// TwinCAT 3 PLC project Base
// ProgramVersion: 3.1.4022.4
// libraries:
//   Tc2_Standard, * (Beckhoff Automation GmbH)
//   Tc2_System, * (Beckhoff Automation GmbH)
//   Tc2_Utilities, * (Beckhoff Automation GmbH)
//   Tc3_IotCommunicator, * (Beckhoff Automation GmbH)
//   Tc3_JsonXml, * (Beckhoff Automation GmbH)
//   Tc3_Module, * (Beckhoff Automation GmbH)
// project tree:
//   DUTs/ E_JsonStates.TcDUT (not stored)
//   GVLs/ CELL_STATE.TcGVL (not stored), CELL_WORKING_STATES.TcGVL (not stored), CLAMP_STATE.TcGVL (not stored), CELL_ACTION_STATE.TcGVL, DATA_SERVICE_STATE.TcGVL (not stored), MHS_STATE.TcGVL
//   / PlcTask.TcTTO
//   POUs/ FB_VirtualCell.TcPOU, I_CELL.TcIO, FB_Cell.TcPOU, FB_Clamp.TcPOU, FB_ClampSimulated.TcPOU (not stored), FB_DataService.TcPOU, FB_InterfaceIO.TcPOU, FB_InterfaceSimulated.TcPOU (not stored), FB_MHS.TcPOU, ITF_Cell.TcIO (not stored), JsonSaxHandler.TcPOU (not stored), MAIN.TcPOU, POU.TcPOU, FB_VirtualCellIntWriter.TcPOU (not stored)
// real-time tasks:
//   TASK PlcTask: cycle T#10ms, priority 20, ADS port 350

CONFIGURATION Base
    RESOURCE PLC ON TwinCAT3
        TASK PlcTask(INTERVAL := T#10ms, PRIORITY := 20);
        PROGRAM MAIN WITH PlcTask : MAIN;
    END_RESOURCE
END_CONFIGURATION

// ---- GVLs/CELL_ACTION_STATE.TcGVL
{attribute 'qualified_only'}
VAR_GLOBAL
			
TYPE 
	CELL_ACTION_STATE: (e_ToStandby, e_Standby, e_ToLoadPos, e_LoadPos, e_ToStartabel, e_Startabel, e_ToRunning , e_Running, 
				e_ToUnLoadPos, e_UnLoadPos,e_Finished, e_ToEmergencyStop, e_EmergencyStop, e_ToEmergencyOff, e_EmergencyOff , e_ErrorNum);
	
	
				
END_TYPE


END_VAR

// ---- GVLs/MHS_STATE.TcGVL
{attribute 'qualified_only'}
VAR_GLOBAL
TYPE
	MHS_STATE: (e_IDLE, e_PGO_POS, e_PGET_WP, e_PWAIT_DOOR, e_PWAIT_CLAMP, e_PPUT_WP,e_PCLOSE_CLAMP , e_PLEAFE_MACHINE, 
				e_GGO_POS, e_GGET_WP, e_GWAIT_DOOR, e_GWAIT_CLAMP ,e_GCLOSE_CLAMP , e_GLEAFE_MACHINE, e_AKTION_FINISHED, e_ERROR);
END_TYPE	

END_VAR

// ---- POUs/I_CELL.TcIO
INTERFACE I_CELL

METHOD GetErrorString : STRING
VAR_INPUT
END_VAR
END_METHOD

METHOD GetName : STRING
VAR_INPUT
END_VAR
END_METHOD

METHOD GetState : INT
VAR_INPUT
END_VAR
END_METHOD

METHOD GetWorkpiece : DINT
VAR_INPUT
END_VAR
END_METHOD

METHOD IsDisassemblyCell : BOOL
VAR_INPUT
END_VAR
END_METHOD

METHOD IsError : BOOL
VAR_INPUT
END_VAR
END_METHOD

METHOD IsIdle : BOOL
VAR_INPUT
END_VAR
END_METHOD

METHOD IsVirtualCell : BOOL
VAR_INPUT
END_VAR
END_METHOD

METHOD RequestActionState : BOOL
VAR_INPUT
	csStateRequest : CELL_ACTION_STATE;
END_VAR
END_METHOD

METHOD RequestWork : BOOL
VAR_INPUT
END_VAR
END_METHOD

METHOD SetDisassemblyCell : BOOL
VAR_INPUT
	bIsDisassemblyCell : BOOL;
END_VAR
END_METHOD

METHOD SetGetDataServiceEnable : BOOL
VAR_INPUT
END_VAR
END_METHOD

METHOD SetName : BOOL
VAR_INPUT
	sName :string ;
END_VAR
END_METHOD

METHOD SetPutDataServiceEnable : BOOL
VAR_INPUT
END_VAR
END_METHOD

METHOD SetVirtualCell : BOOL
VAR_INPUT
END_VAR
END_METHOD

METHOD SetWorkpiece : BOOL
VAR_INPUT
	iWorkpiece : DINT;
	sWorkpieceID : STRING;
END_VAR
END_METHOD

METHOD StateMachine : BOOL
VAR_INPUT
END_VAR
END_METHOD

END_INTERFACE

// ---- POUs/MAIN.TcPOU

PROGRAM MAIN
	
VAR



// Allg. nitwendige Variablen
m_bInit : BOOL;
I : DINT;
sString : STRING;
diDint : DINT;
bBOOL:BOOL;
m_iCellUpdateIter : INT := 0; // Iterationsvariable für die Json Strings der Zelle

// Zellen
fbCellA2 : FB_Cell;
fbCellB2 : FB_Cell; 
fbCellB5 : FB_Cell; 
fbCellV1 : FB_VirtualCell;
fbCellV2 : FB_VirtualCell;

aCellList : ARRAY [1..5] OF I_CELL; // Liste der Zellen
m_iNumberOfCells : DINT := 5; // Bei hinzufügen/löschen einer Zelle ist hier die Anzahl anzupassen

// MHS 
fbMHS : FB_MHS;

// Kommunikations-Variabeln für Aktionen von der GUI


m_bTrigger : BOOL;// Trigger zum zyklischen Aktualisieren der Anwendung
m_iTriggerTimer : INT; // Zähler zum Trigger 
m_sJsonTrigger : STRING(80);

m_sActionID : STRING(80);
m_sWPID : STRING(80);
m_iWPRequest : DINT;
m_sCellRequest : STRING;
m_iActionRequest : DINT;
m_iActionState : DINT;


m_sActionIDLast : STRING(80);
m_sWPIDLast : STRING(80);
m_iWPRequestLast : DINT;
m_iCellRequestLast : DINT;
m_iActionRequestLast : DINT;
m_iActionStateLast : DINT;
m_iCellRequest : DINT;

m_bAktionInProgress : BOOL; 

//JSON-Variablen
	//Writer
	m_iJsonTimer 		: DINT;
 	dtTimestamp 		: DATE_AND_TIME := DT#2017-04-04-12:42:42;
 	fbJson      		: FB_JsonSaxWriter;
 	sJsonDocCells   	: STRING(3000);
	//Reader
 	fbJsonReader    		: FB_JsonSaxReader;
	pJsonParse 				: JsonSaxHandler;
	sJsonDocAction			: STRING(255);
	sJsonDocLastAction   : STRING(255);
	
	sJsonDocError 		 : STRING (255); 

END_VAR


//Initialisierung
IF NOT m_bInit THEN
	// Hier die FunktionsBlöcke der Maschinen in das Array Schreiben !!!
	aCellList[1] := fbCellA2;
	aCellList[1].SetName('A2'); // Geometrieerfassung
	//aCellList[1].SetPutDataServiceEnable();
	aCellList[2] := fbCellB2;
	aCellList[2].SetName('B2'); // Rekonturierng
 	aCellList[2].SetGetDataServiceEnable();
	aCellList[3] := fbCellB5;
	aCellList[3].SetName('B5'); // LaserSchweißen
	aCellList[3].SetGetDataServiceEnable();
	aCellList[3].SetPutDataServiceEnable();
	
	aCellList[4] := fbCellV1;
	aCellList[4].SetName('V1'); // Virtuell
	aCellList[4].SetVirtualCell();
	
	
	aCellList[5] := fbCellV2;
	aCellList[5].SetName('V2'); // Virtuell
	aCellList[5].SetVirtualCell();

	// Intitialisiert setzen 
	m_bInit := TRUE;

END_IF



IF m_bAktionInProgress = FALSE THEN 
	// Abfrage ob neue Aktion angestoßen wurde
	CheckForNewAction();
		
END_IF


//Zustandmaschinen
	// Zyklische aktualisierung der Zellen-Zustandsmaschinen
	I := 1;
	FOR I:=1 TO m_iNumberOfCells BY 1 DO
    	aCellList[I].StateMachine();
	END_FOR;
	// Zyklische aktualisierung der MHS-Zustandsmaschine
	fbMHS();
// Zustandsmaschinen durchgelaufen

IF m_bAktionInProgress THEN// MHS muss den Zustand der involvierten Zelle kennen und eine Zustand von der Zelle anfordern können
	
	fbMHS.SetStateCurrentMachineForAction( aCellList[fbMHS.GetCurrentCellForAction()].GetState());// Aktualisieren des MHS Zustandes
	IF fbMHS.NeededCellStatePending() THEN // Wenn das MHS einen Zellenzustand verlangt wird er folgend übergeben
		aCellList[fbMHS.GetCurrentCellForAction()].RequestActionState(fbMHS.SendNeededToCell() );// Übergabe des geforderten Zellenzustandes an die Zelle
	END_IF
END_IF


// Abfrage ob letzte Aktion Abgeschlossen wurde.... auf WIN abgefragen um neue Aktion zu senden 
IF fbMHS.GetActionFinished() THEN
	m_bAktionInProgress := FALSE; 
	IF m_iActionRequestLast = 2 THEN // Bestuecken
		aCellList[m_iCellRequestLast].SetWorkpiece(m_iWPRequestLast, m_sWPIDLast);// Werkstück an die Zelle übergeben
		aCellList[m_iCellRequestLast].RequestWork(); // Starten der Bearbeitung in der Zelle		
	ELSE
		aCellList[m_iCellRequestLast].SetWorkpiece(0, 'Empty'); // Werkstück der Zelle nehmen
	END_IF
	m_iActionStateLast := 3;
END_IF

// Schreiben der JSON-Strings zur Kommunikation der Systemdemostrator-Anwendung
WriteJsonStrings();

METHOD CheckForNewAction : BOOL
VAR_INPUT
END_VAR
	 ParseNewAction();
	m_iCellRequest := NumberOfCellName(m_sCellRequest);
	IF	 (NOT(m_sActionID = m_sActionIDLast)) AND (m_iCellRequest <= m_iNumberOfCells) AND (m_iCellRequest > 0) THEN // Neue Aktion und Zelle ist existent
		IF NOT(aCellList[m_iCellRequest].IsVirtualCell())THEN
			
			IF aCellList[m_iCellRequest].IsIdle() THEN // Zelle frei
				// Neue Aktion an das MHS übergeben 
				WriteNewActionToMHS();
				m_bAktionInProgress := TRUE;// Setzen des Flags 
			END_IF
		ELSE // Im Falle einer Aktion für eine virtuelle Zelle
			IF aCellList[m_iCellRequest].IsIdle() THEN
				aCellList[m_iCellRequest].SetWorkpiece(0, m_sWPID );
				aCellList[m_iCellRequest].RequestWork();	
				//m_iActionStateLast := 3; // Wird nur angestoßen ist direkt fertig mit der Aktion, so dass eine weitere beginnen kann.
			END_IF
		END_IF
	
	END_IF
END_METHOD

METHOD NumberOfCellName : DINT
VAR_INPUT
	sNameOfCell : STRING;
END_VAR
FOR I:=1 TO m_iNumberOfCells BY 1 DO
    IF sNameOfCell = aCellList[I].GetName() THEN
		NumberOfCellName :=I;
	END_IF
END_FOR;
END_METHOD

METHOD ParseNewAction : BOOL
VAR_INPUT
END_VAR

	// Aktion JSonDoc Lesen des Aktuellen Strings
	fbJsonReader.Parse( sJson := sJsonDocAction, ipHdl := pJsonParse);
	
	IF pJsonParse.IsFinished() THEN
		// Übergabe der geparsten Variablen
		m_sActionID	:=	pJsonParse.GetActionID();
		m_sWPID	:=	pJsonParse.GetWPID();
		m_iWPRequest := pJsonParse.GetWPPlace(); 
		m_sCellRequest := pJsonParse.GetCell(); 
		m_iActionRequest:=pJsonParse.GetActionType();
		
		// Für den nächsten Durchlauf zurücksetzen 
		pJsonParse.Reset();
	ELSE
		// Parsen des Json-Strings
		fbJsonReader.Parse( sJson := sJsonDocAction, ipHdl := pJsonParse);
	END_IF
END_METHOD

METHOD WriteJSonDocAction : BOOL
VAR_INPUT
END_VAR

fbJson.ResetDocument();
		//fbJson.StartArray();
fbJson.StartObject();
            fbJson.AddKey('m_sActionID');
			fbJson.AddString(m_sActionIDLast);
            fbJson.AddKey('m_sWPID');
			sString := m_sWPIDLast;
			fbJson.AddString(sString);
            fbJson.AddKey('m_iWPPlace');
			fbJson.AddDint(m_iWPRequestLast);
            fbJson.AddKey('m_sCell');
			IF m_iCellRequestLast > 0 THEN// Sonst würden das Zell Array außerhalb seines Bereiches angesproehcen werden
				sString := aCellList[m_iCellRequestLast].GetName();
			ELSE
				sString := 'EmptyAction';				
			END_IF
			fbJson.AddString(sString);
            fbJson.AddKey('m_eActionType');
			fbJson.AddDint(m_iActionRequestLast);
            fbJson.AddKey('m_iActionState');
			fbJson.AddDint(m_iActionStateLast);	
fbJson.EndObject();
	sJsonDocLastAction := fbJson.GetDocument();

WriteJSonDocAction := TRUE;
END_METHOD

METHOD WriteJSonDocCells : BOOL
VAR_INPUT
END_VAR
// Merken alle Zellen einzelnd Updaten, weil es nicht möglich ist die über 255 Zeichen langen Strings aller zu übertragen

	fbJson.ResetDocument();
	//fbJson.StartObject();
	//fbJson.AddKey('Timestamp');
	
	//fbJson.AddDateTime(dtTimestamp);
	m_iCellUpdateIter := m_iCellUpdateIter +1 ; 
	IF m_iCellUpdateIter > m_iNumberOfCells THEN
		m_iCellUpdateIter := 1;
	END_IF
		//fbJson.AddKey('Cell');
		m_sActionIDLast := m_sActionID;
		m_iWPRequestLast := m_iWPRequest; 		
		m_iCellRequestLast := m_iCellRequest;
		m_iActionRequestLast :=	m_iActionRequest;
		fbJson.StartObject();
		//fbJson.StartArray();
		fbJson.AddKey('Name');
		sString := aCellList[m_iCellUpdateIter].GetName();
		fbJson.AddString(sString);
		fbJson.AddKey('State');
		fbJson.AddDint(aCellList[m_iCellUpdateIter].GetState());
		fbJson.AddKeyBool('Idle',aCellList[m_iCellUpdateIter].IsIdle());
		fbJson.AddKey('Workpiece');
		fbJson.AddDint(aCellList[m_iCellUpdateIter].GetWorkpiece());
		fbJson.AddKey('IsDisassemblyCell');
		fbJson.AddBool(aCellList[m_iCellUpdateIter].IsDisassemblyCell());
		fbJson.AddKey('IsVirtualCell');
		fbJson.AddBool(aCellList[m_iCellUpdateIter].IsVirtualCell());
		fbJson.EndObject();
		
		

	
	
	//fbJson.EndObject();
	sJsonDocCells := '';
	sJsonDocCells := fbJson.GetDocument();
	
WriteJSonDocCells := TRUE;
END_METHOD

METHOD WriteJSonError : BOOL
VAR_INPUT
END_VAR
	fbJson.ResetDocument();


	I := 1;
	FOR I:=1 TO m_iNumberOfCells BY 1 DO
		IF aCellList[I].IsError() THEN
			fbJson.StartObject();
			fbJson.AddKey('Name');
			sString := aCellList[I].GetName();
			fbJson.AddString(sString);	
			fbJson.AddKey('Workpiece');
			fbJson.AddDint(aCellList[I].GetWorkpiece());
			fbJson.AddKey('Error');
			sString := aCellList[I].GetErrorString();
			fbJson.AddString(sString);
			fbJson.EndObject();	
			
			sJsonDocError := '';
			sJsonDocError := fbJson.GetDocument();

		END_IF	
	
	END_FOR;
END_METHOD

METHOD WriteJsonStrings : BOOL
VAR_INPUT
END_VAR




// Erstellen eines Json-Strings für die GUI alle 100 Durchläufe 0,1s
m_iJsonTimer := m_iJsonTimer+1;
IF m_iJsonTimer > 150 THEN
	WriteJSonDocCells();
	WriteJSonDocAction();
	
	m_iJsonTimer := 0;
	
END_IF
// GUI Trigger um zyklische Aufrufe auch bei nicht veränderten JSON-Strings zu erzielen
// Ohne den Trigger würde ine Prüfung des Regenerationspfades bei nicht mehr vorhanden Aktion im Pfad nicht fortgeführt werden
IF m_iTriggerTimer > 2500 THEN
	m_bTrigger :=  NOT(m_bTrigger);// Bool abwechselnd false und true
	WriteJsonTrigger();
	m_iTriggerTimer := 0; 
END_IF
	
m_iTriggerTimer := m_iTriggerTimer + 1;
END_METHOD

METHOD WriteJsonTrigger : BOOL
VAR_INPUT
END_VAR
fbJson.ResetDocument();
		//fbJson.StartArray();
fbJson.StartObject();
            fbJson.AddKey('m_bTrigger');
			fbJson.AddBool(m_bTrigger);
fbJson.EndObject();
	m_sJsonTrigger := fbJson.GetDocument();
END_METHOD

METHOD WriteNewActionToMHS : BOOL
VAR_INPUT
END_VAR
// Übergaben der neuen Aktion an das MHS
fbMHS.RequestAction(	iWorkpiece := m_iWPRequest, iCell := m_iCellRequest, bRequest := m_iActionRequest);
// Speichern des Zustandes
m_sActionIDLast := m_sActionID;
m_sWPIDLast := m_sWPID; 
m_iWPRequestLast := m_iWPRequest; 		
m_iCellRequestLast := m_iCellRequest;
m_iActionRequestLast :=	m_iActionRequest;

m_iActionStateLast := 2;
END_METHOD

END_PROGRAM

// ---- POUs/FB_Cell.TcPOU
FUNCTION_BLOCK FB_Cell IMPLEMENTS I_CELL
VAR_INPUT
	
END_VAR
VAR_OUTPUT
END_VAR
VAR
	m_csStateRequest : CELL_ACTION_STATE;
	m_csStateRequestOld : CELL_ACTION_STATE;
	m_csState : CELL_ACTION_STATE;
	m_csStateLastCycle : CELL_ACTION_STATE;
	m_csStateLastAction : CELL_ACTION_STATE;
	
	
	m_csSRWorkingState : CELL_WORKING_STATES := CELL_WORKING_STATES.e_FINISHED;
	m_csSRWorkingStateLast : CELL_WORKING_STATES := CELL_WORKING_STATES.e_FINISHED;
	// Eigenschaften
	m_sName : STRING;
	m_bIsDisassemblyCell : BOOL;
	
	
	m_iWorkpiece : DINT;
	m_sWorkpieceID : STRING;
	

	m_csCellState : CELL_STATE;
	m_csCellStateLast : CELL_STATE;

	fbInterface : FB_InterfaceSimulated;
	fbClamp : FB_ClampSimulated; 
	
	m_sErrorString : STRING;
	
	// DataServices
	
	fbDataServicePut : FB_DataService;
	m_bDataServicePutEnable : BOOL;
	fbDataServiceGet : FB_DataService;
	m_bDataServiceGetEnable : BOOL;
	m_sConfigString : STRING;
	m_sConfigStringEndGet : STRING  := '_Get.exe';
	m_sConfigStringEndPut : STRING  := '_Put.exe';
	m_sDataServiceDir: STRING  := 'C:\temp\Debug\';
	m_sDataServiceIP: STRING  := '192.168.178.24.1.1';
	
END_VAR

METHOD GetErrorString : STRING
VAR_INPUT
END_VAR
END_METHOD

METHOD GetName : STRING
VAR_INPUT
END_VAR
GetName := m_sName;
END_METHOD

METHOD PUBLIC GetState : INT
VAR_INPUT
	
END_VAR
GetState := m_csState;
END_METHOD

METHOD GetWorkpiece : DINT
VAR_INPUT
END_VAR
GetWorkpiece := m_iWorkpiece;
END_METHOD

METHOD IsDisassemblyCell : BOOL
VAR_INPUT
END_VAR
IsDisassemblyCell := m_bIsDisassemblyCell;
END_METHOD

METHOD IsError : BOOL
VAR_INPUT
END_VAR
IF m_csCellState = CELL_STATE.e_ERROR THEN
	IsError := TRUE;
END_IF
END_METHOD

METHOD IsIdle : BOOL
VAR_INPUT
END_VAR
IF m_csCellState = CELL_STATE.e_IDEL THEN
	IsIdle := TRUE;
END_IF
END_METHOD

METHOD IsVirtualCell : BOOL
VAR_INPUT
END_VAR
IsVirtualCell :=FALSE;
END_METHOD

METHOD PUBLIC RequestActionState : BOOL
VAR_INPUT
	csStateRequest : CELL_ACTION_STATE;
END_VAR
m_csStateRequest := csStateRequest;
END_METHOD

METHOD RequestWork : BOOL
VAR_INPUT
END_VAR
m_csCellState := CELL_STATE.e_WORKING;
END_METHOD

METHOD SetDisassemblyCell : BOOL
VAR_INPUT
	bIsDisassemblyCell : BOOL;
END_VAR
m_bIsDisassemblyCell := bIsDisassemblyCell;
END_METHOD

METHOD SetGetDataServiceEnable : BOOL
VAR_INPUT
END_VAR
m_bDataServiceGetEnable := TRUE;
SetGetDataServiceEnable := TRUE;
END_METHOD

METHOD SetName : BOOL
VAR_INPUT
	sName :string ;
END_VAR
m_sName := sName;
END_METHOD

METHOD SetPutDataServiceEnable : BOOL
VAR_INPUT
END_VAR
m_bDataServicePutEnable := TRUE;
SetPutDataServiceEnable := TRUE;
END_METHOD

METHOD SetVirtualCell : BOOL
VAR_INPUT
END_VAR
END_METHOD

METHOD SetWorkpiece : BOOL
VAR_INPUT
	iWorkpiece : DINT;
	sWorkpieceID : STRING;
END_VAR
m_iWorkpiece := iWorkpiece;
m_sWorkpieceID := sWorkpieceID;
END_METHOD

METHOD PUBLIC StateMachine : BOOL
VAR_INPUT
END_VAR

fbInterface();
fbClamp();



// Error-Abfragen
IF fbClamp.IsError() THEN
	m_csCellState := CELL_STATE.e_ERROR; 
	m_sErrorString := 'CLAMP-Error: Clamp is closed without Workpiece';
END_IF


//Zellen Zustandsmaschine

CASE m_csCellState OF 
	CELL_STATE.e_IDEL:
			
	
		;
 	CELL_STATE.e_MHS_ACTION;
		//SubRoutine für Aktion beim beladen aktuell leer da alles vom MHS gesteuert wird 
	
		;
	CELL_STATE.e_WORKING:
		//SubRoutine zum Durchführen einer Bearbeitung
		
		IF NOT (m_csCellStateLast = m_csCellState) THEN
			m_csSRWorkingState := CELL_WORKING_STATES.e_START;
			IF m_bDataServiceGetEnable THEN
				fbDataServiceGet.SetNetIP(m_sDataServiceIP);
				fbDataServiceGet.SetWorkingDirectory(m_sDataServiceDir);
				m_sConfigString := m_sDataServiceDir;
				m_sConfigString := CONCAT(m_sConfigString , m_sName); // erstellen des Pfades der Applikation 
				m_sConfigString := CONCAT(m_sConfigString , m_sConfigStringEndGet);
				fbDataServiceGet.SetCommandLine(m_sWorkpieceID);
				fbDataServiceGet.SetPathOfApplication(m_sConfigString);
				fbDataServiceGet.StartDataService();
			END_IF
		END_IF
			
		CASE m_csSRWorkingState OF
			
			CELL_WORKING_STATES.e_START:
				
				IF NOT (m_csSRWorkingStateLast = m_csSRWorkingState )THEN
					m_csStateRequest := CELL_ACTION_STATE.e_Startabel;
				END_IF
				
				
				IF m_csState = CELL_ACTION_STATE.e_Startabel AND (fbDataServiceGet.IsFinished() OR NOT(m_bDataServiceGetEnable) )  THEN // Zelle bereit zum Starten und DataServiceGet fertig oder nicht konfiguriert
					m_csSRWorkingState:= CELL_WORKING_STATES.e_WORKING;
					fbDataServiceGet.SetIdle();
					m_csStateRequest:= CELL_ACTION_STATE.e_Running;
				END_IF
				
				
			CELL_WORKING_STATES.e_WORKING:
				IF NOT (m_csSRWorkingStateLast = m_csSRWorkingState) THEN
					m_csStateRequest := CELL_ACTION_STATE.e_Running;
				END_IF
				
				IF m_csState = CELL_ACTION_STATE.e_Finished THEN
					m_csSRWorkingState := CELL_WORKING_STATES.e_FINISHED;
					IF m_bDataServicePutEnable THEN
						fbDataServicePut.SetNetIP('192.168.178.24.1.1');
						fbDataServicePut.SetWorkingDirectory('C:\temp\Debug');
						m_sConfigString := 'C:\temp\Debug\';						
						m_sConfigString := CONCAT(m_sConfigString , m_sName); // erstellen des Pfades der Applikation 
						m_sConfigString := CONCAT(m_sConfigString , m_sConfigStringEndPut);// erstellen des Pfades der Applikation
						fbDataServicePut.SetCommandLine(m_sWorkpieceID);
						fbDataServicePut.SetPathOfApplication(m_sConfigString);
						fbDataServicePut.StartDataService();
						m_csSRWorkingState := e_DATAPUT;
					END_IF
		
				END_IF
			CELL_WORKING_STATES.e_DATAPUT:
					IF fbDataServicePut.IsFinished() THEN
						fbDataServicePut.SetIdle();
						m_csSRWorkingState := CELL_WORKING_STATES.e_FINISHED;
					END_IF
					IF fbDataServicePut.IsError() THEN
						fbDataServicePut.SetIdle();
						m_csSRWorkingState := CELL_STATE.e_ERROR;
					END_IF
					
			CELL_WORKING_STATES.e_FINISHED:
				m_csCellState := CELL_STATE.e_IDEL;
			
		END_CASE
		
		
		
	CELL_STATE.e_ERROR:
		m_csState :=CELL_ACTION_STATE.e_ToEmergencyStop;
	
		
END_CASE
m_csSRWorkingStateLast := m_csSRWorkingState;
m_csCellStateLast := m_csCellState;

IF NOT (m_csStateRequestOld = m_csStateRequest) THEN
	m_csState := m_csStateRequest - 1;
	m_csStateRequestOld := m_csStateRequest;
END_IF


// Aktions Zustandsmaschine
CASE m_csState OF 
	CELL_ACTION_STATE.e_ToStandby:
		IF NOT (m_csStateLastCycle = m_csState) THEN
			fbInterface.SetStandby(TRUE);
			m_csStateLastAction := m_csStateLastCycle;
		END_IF
		
		IF fbInterface.GetStandby() THEN
			m_csState := e_Standby; 
		END_IF
		
	CELL_ACTION_STATE.e_Standby :
	
		IF NOT (m_csStateLastCycle = m_csState) THEN
			m_csStateLastAction := m_csStateLastCycle;
		END_IF
		fbInterface.SetStandby(FALSE);
		
	CELL_ACTION_STATE.e_ToLoadPos:
	
		IF NOT (m_csStateLastCycle = m_csState) THEN
			m_csStateLastAction := m_csStateLastCycle;
			fbInterface.SetMoveToLoad(TRUE);
			fbClamp.SetOpenClamp();
		END_IF
		
		IF fbInterface.GetLoadPos() AND fbClamp.IsOpen() THEN
			m_csState := e_LoadPos; 
		END_IF
		
		
	CELL_ACTION_STATE.e_LoadPos:
	
		IF NOT (m_csStateLastCycle = m_csState) THEN
			m_csStateLastAction := m_csStateLastCycle;
		END_IF
		fbInterface.SetMoveToLoad(FALSE);
				
		
	CELL_ACTION_STATE.e_ToStartabel:
	
		IF NOT (m_csStateLastCycle = m_csState) THEN
			m_csStateLastAction := m_csStateLastCycle;
			fbClamp.SetCloseClampFull();
		END_IF
		
		
		IF  fbClamp.IsClosedFull() THEN //fbInterface.GetStartable() AND
			m_csState := e_Startabel; 
		END_IF
		
	CELL_ACTION_STATE.e_Startabel:
	
		IF NOT (m_csStateLastCycle = m_csState) THEN
			m_csStateLastAction := m_csStateLastCycle;
			
		END_IF
		
	CELL_ACTION_STATE.e_ToRunning:
	
		IF NOT (m_csStateLastCycle = m_csState) THEN
			m_csStateLastAction := m_csStateLastCycle;
			fbInterface.SetStart(TRUE);
		END_IF
		
		IF fbInterface.GetIsRunning() THEN
			m_csState := CELL_ACTION_STATE.e_Running; 
		END_IF
		
	CELL_ACTION_STATE.e_Running:
	
		IF NOT (m_csStateLastCycle = m_csState) THEN
			m_csStateLastAction := m_csStateLastCycle;
		END_IF
		fbInterface.SetStart(FALSE);
		IF fbInterface.GetFinished() THEN
			m_csState := CELL_ACTION_STATE.e_Finished;		
		END_IF
	CELL_ACTION_STATE.e_Finished:
		IF NOT (m_csStateLastCycle = m_csState) THEN
			m_csStateLastAction := m_csStateLastCycle;
		END_IF
		
	CELL_ACTION_STATE.e_ToUnLoadPos:
 
		IF NOT (m_csStateLastCycle = m_csState) THEN
			m_csStateLastAction := m_csStateLastCycle;
			fbClamp.SetOpenClamp();
		END_IF
		
		
		IF fbInterface.GetUnloadPos() AND fbClamp.IsOpen() THEN
			m_csState := e_UnLoadPos; 
		END_IF
		
	CELL_ACTION_STATE.e_UnLoadPos:
	
		IF NOT (m_csStateLastCycle = m_csState) THEN
			m_csStateLastAction := m_csStateLastCycle;
		END_IF
		
	CELL_ACTION_STATE.e_ToEmergencyStop:
	
		IF NOT (m_csStateLastCycle = m_csState) THEN
			m_csStateLastAction := m_csStateLastCycle;
		END_IF
		
		
		IF fbInterface.GetEmergencyStop() THEN
			m_csState := e_EmergencyStop; 
		END_IF
		
	CELL_ACTION_STATE.e_EmergencyStop:
	
		IF NOT (m_csStateLastCycle = m_csState) THEN
			m_csStateLastAction := m_csStateLastCycle;
		END_IF
		
	CELL_ACTION_STATE.e_ToEmergencyOff:
	
		IF NOT (m_csStateLastCycle = m_csState) THEN
			m_csStateLastAction := m_csStateLastCycle;
		END_IF
		
		
		IF fbInterface.GetEmergencyStop() THEN
			m_csState := e_EmergencyOff; 
		END_IF
		
	CELL_ACTION_STATE.e_EmergencyOff:
	
		IF NOT (m_csStateLastCycle = m_csState) THEN
			m_csStateLastAction := m_csStateLastCycle;
		END_IF
		
	ELSE
		IF NOT (m_csStateLastCycle = m_csState) THEN
			m_csStateLastAction := m_csStateLastCycle;
		END_IF
		
END_CASE

IF m_bDataServiceGetEnable THEN
	fbDataServiceGet();
END_IF
IF m_bDataServicePutEnable THEN	
	fbDataServicePut();
END_IF

m_csStateLastCycle := m_csState;
END_METHOD

END_FUNCTION_BLOCK

// ---- POUs/FB_DataService.TcPOU
FUNCTION_BLOCK FB_DataService
VAR_INPUT
END_VAR
VAR_OUTPUT
END_VAR
VAR
	fbStartProcess : NT_StartProcess;

	m_sCommandLine : STRING;
	m_sNetIP : STRING;
	m_sWorkingdirektory : STRING;
	m_sPathOfApplication : STRING;
	m_bStart : BOOL;
	m_eState : DATA_SERVICE_STATE;
	m_sErrCode : STRING;
	m_iReturnValue : DINT;
END_VAR

fbStartProcess.NETID 		:= m_sNetIP; // IP Adresse des Rechners auf dem die Zwillinge liegen
fbStartProcess.COMNDLINE 	:= m_sCommandLine; // Hier muss die ZwillingsID/ ProjektID übertragen werden
fbStartProcess.DIRNAME 		:= m_sWorkingdirektory; // Dieser Verzeichnis ist  vermutlich immer c:\TEMP
fbStartProcess.PATHSTR 		:= m_sPathOfApplication; // Pfad direkt zur DataService.exe wobei sich diese aus dem Zell-Namen ergibt 


IF fbStartProcess.ERR THEN // Fehlerabrage bereits vor der Zustandsmaschine 
	m_eState := DATA_SERVICE_STATE.e_ERROR;
END_IF 


CASE m_eState OF 
	DATA_SERVICE_STATE.e_IDLE:
	
		IF  m_bStart = TRUE THEN
			fbStartProcess.START := TRUE;
			m_bStart := FALSE; //Nurpositive Flanke übergeben		
		END_IF
	
		IF fbStartProcess.BUSY = TRUE THEN // Wenn der Funktionsblock selber Busy meldet in den nächsten Zustand
			m_eState := DATA_SERVICE_STATE.e_BUSY;
			fbStartProcess.START := FALSE;  
		END_IF
		
	DATA_SERVICE_STATE.e_BUSY:
	
 		IF fbStartProcess.BUSY = FALSE THEN
			IF m_iReturnValue = 1 THEN // Übergabewert der DataService.exe
				m_iReturnValue := 0; // Zurücksetzen für den nächsten Durchlauf
				m_eState := DATA_SERVICE_STATE.e_FINISHED;
			END_IF
			IF m_iReturnValue = 2 THEN
				m_eState := DATA_SERVICE_STATE.e_ERROR; 					
			END_IF		
		END_IF 
		
	DATA_SERVICE_STATE.e_FINISHED: // Zustand erforderlich da somit ein Zyklus lang abgefragt werden kann ob der Ablauf erfolgreich war
			
 		
		
	DATA_SERVICE_STATE.e_ERROR:
	
		m_sErrCode := UDINT_TO_STRING (fbStartProcess.ERRID); // Der Fehler wird als ganzzahl in den String geschrieben 
	
ELSE // Sicherheit bei falschem Wert
		m_eState := DATA_SERVICE_STATE.e_ERROR;
		m_sErrCode := 'Falscher Wert DataService-Status nicht vorhanden';
		
END_CASE

// Aufruf des Funktionblocks NT_StartProcess
fbStartProcess();

METHOD GetErrorCode : STRING
VAR_INPUT
END_VAR

VAR
END_VAR
GetErrorCode :=m_sErrCode;
END_METHOD

METHOD IsBusy : BOOL
VAR_INPUT
END_VAR
IF m_eState = DATA_SERVICE_STATE.e_BUSY THEN
	IsBusy := TRUE;
END_IF
END_METHOD

METHOD IsError : BOOL
VAR_INPUT
END_VAR
IF m_eState = DATA_SERVICE_STATE.e_ERROR THEN
	IsError := TRUE;
END_IF
END_METHOD

METHOD IsFinished : BOOL
VAR_INPUT
END_VAR
IF m_eState = DATA_SERVICE_STATE.e_FINISHED THEN
	IsFinished := TRUE;
END_IF
END_METHOD

METHOD IsIdle : BOOL
VAR_INPUT
END_VAR
IF m_eState = DATA_SERVICE_STATE.e_IDLE THEN
	IsIdle := TRUE;
END_IF
END_METHOD

METHOD SetCommandLine : BOOL
VAR_INPUT
	sCommandLine : STRING;
END_VAR
m_sCommandLine := sCommandLine;
END_METHOD

METHOD SetIdle : BOOL
VAR_INPUT
END_VAR
m_eState := DATA_SERVICE_STATE.e_IDLE;
END_METHOD

METHOD SetNetIP : BOOL
VAR_INPUT
	sNetIP : STRING;
END_VAR
m_sNetIP := sNetIP;
END_METHOD

METHOD SetPathOfApplication : BOOL
VAR_INPUT
	sPathOfApplication :STRING;
END_VAR
 m_sPathOfApplication := sPathOfApplication;
END_METHOD

METHOD SetWorkingDirectory : BOOL
VAR_INPUT
	sWorkingdirektory : STRING;
END_VAR
m_sWorkingdirektory := sWorkingdirektory;
END_METHOD

METHOD StartDataService : BOOL
VAR_INPUT
END_VAR
m_bStart := TRUE;
StartDataService := TRUE;
END_METHOD

END_FUNCTION_BLOCK

// ---- POUs/FB_VirtualCell.TcPOU
FUNCTION_BLOCK FB_VirtualCell IMPLEMENTS I_CELL
VAR_INPUT
	
END_VAR
VAR_OUTPUT
END_VAR
VAR
	m_csStateRequest : CELL_ACTION_STATE;
	m_csStateRequestOld : CELL_ACTION_STATE;
	m_csState : CELL_ACTION_STATE;
	m_csStateLastCycle : CELL_ACTION_STATE;
	m_csStateLastAction : CELL_ACTION_STATE;
	
	
	m_csSRWorkingState : CELL_WORKING_STATES := CELL_WORKING_STATES.e_FINISHED;
	m_csSRWorkingStateLast : CELL_WORKING_STATES := CELL_WORKING_STATES.e_FINISHED;
	// Eigenschaften
	m_sName : STRING;
	m_bIsDisassemblyCell : BOOL;
	
	m_iWorkpiece : DINT;
	m_sWorkpieceID : STRING;
	

	m_csCellState : CELL_STATE;
	m_csCellStateLast : CELL_STATE;


	
	m_sErrorString : STRING;
	
	// DataServices
	

	m_sConfigString : STRING;
	m_sConfigStringEndGet : STRING  := '_Get.exe';
	m_sConfigStringEndPut : STRING  := '_Put.exe';
	
	// Virtuelle Zellen Verbindung
	fbVirtualCellIntWriter 	: FB_VirtualCellIntWriter;
	fbJson      			: FB_JsonSaxWriter;
	m_sJsonAction 			: STRING;
	m_sActionPath 			: STRING;
	m_sActionName			: STRING;
	m_sActionPathDir 		: STRING   := 'C:\temp\Actions';
	m_sAMSNetID 			: 	STRING 	:=	'192.168.178.24.1.1';
	
END_VAR

METHOD GetErrorString : STRING
VAR_INPUT
END_VAR
END_METHOD

METHOD GetName : STRING
VAR_INPUT
END_VAR
GetName := m_sName;
END_METHOD

METHOD PUBLIC GetState : INT
VAR_INPUT
	
END_VAR
GetState := CELL_ACTION_STATE.e_Standby;
END_METHOD

METHOD GetWorkpiece : DINT
VAR_INPUT
END_VAR
GetWorkpiece := m_iWorkpiece;
END_METHOD

METHOD IsDisassemblyCell : BOOL
VAR_INPUT
END_VAR
IsDisassemblyCell := FALSE; // Kann keine sein ist virtuell
END_METHOD

METHOD IsError : BOOL
VAR_INPUT
END_VAR
IF m_csCellState = CELL_STATE.e_ERROR THEN
	IsError := TRUE;
END_IF
END_METHOD

METHOD IsIdle : BOOL
VAR_INPUT
END_VAR
IF m_csCellState = CELL_STATE.e_IDEL THEN
	IsIdle := TRUE;
END_IF
END_METHOD

METHOD IsVirtualCell : BOOL
VAR_INPUT
END_VAR
IsVirtualCell :=TRUE;
END_METHOD

METHOD PUBLIC RequestActionState : BOOL
VAR_INPUT
	csStateRequest : CELL_ACTION_STATE;
END_VAR
m_csStateRequest := csStateRequest;
END_METHOD

METHOD RequestWork : BOOL
VAR_INPUT
END_VAR
m_csCellState := CELL_STATE.e_WORKING;
END_METHOD

METHOD SetDisassemblyCell : BOOL
VAR_INPUT
	bIsDisassemblyCell : BOOL;
END_VAR
m_bIsDisassemblyCell := bIsDisassemblyCell;
END_METHOD

METHOD SetGetDataServiceEnable : BOOL
VAR_INPUT
END_VAR

SetGetDataServiceEnable := FALSE;
END_METHOD

METHOD SetName : BOOL
VAR_INPUT
	sName :string ;
END_VAR
m_sName := sName;
END_METHOD

METHOD SetPutDataServiceEnable : BOOL
VAR_INPUT
END_VAR

SetPutDataServiceEnable := FALSE;
END_METHOD

METHOD SetVirtualCell : BOOL
VAR_INPUT
END_VAR
END_METHOD

METHOD SetWorkpiece : BOOL
VAR_INPUT
	iWorkpiece : DINT;
	sWorkpieceID : STRING;
END_VAR
m_iWorkpiece := iWorkpiece;
m_sWorkpieceID := sWorkpieceID;
END_METHOD

METHOD PUBLIC StateMachine : BOOL
VAR_INPUT
END_VAR

//Zellen Zustandsmaschine

CASE m_csCellState OF 
	CELL_STATE.e_IDEL:
			
	
		;
 	CELL_STATE.e_MHS_ACTION;
		//SubRoutine für Aktion beim beladen aktuell leer da keine MHS für eine virtuelle Zelle verfügbar sind 
		;
	CELL_STATE.e_WORKING:
		//SubRoutine zum Durchführen einer Bearbeitung
			//Erstellen des Json-Strings für die Datei		
			fbJson.ResetDocument();
		
			fbJson.StartObject();
            fbJson.AddKey('Name');
			fbJson.AddString(m_sName);
			fbJson.AddKey('WPID');
			fbJson.AddString(m_sWorkpieceID);			
			fbJson.EndObject();
			m_sJsonAction := fbJson.GetDocument();
		
			// Phad der Schnittstellen-Datei
			m_sActionPath := CONCAT (m_sActionPathDir,'\');
			m_sActionPath := CONCAT (m_sActionPath, m_sName);
			m_sActionPath := CONCAT (m_sActionPath, '_');
			m_sActionPath := CONCAT (m_sActionPath, m_sWorkpieceID);
			m_sActionPath := CONCAT (m_sActionPath, '.json');
			
			// Name der Schnittstellen-Datei
			m_sActionName := CONCAT (m_sName, '_');
			m_sActionName := CONCAT (m_sActionName, m_sWorkpieceID);
			m_sActionName := CONCAT (m_sActionName, '.json');
			
			// Nächster Schritt SubRoutine Starten um das Schreiben auszugühren
			IF NOT (CELL_STATE.e_WORKING = m_csCellStateLast) THEN  
				m_csSRWorkingState := CELL_WORKING_STATES.e_START;
			END_IF

			
	CASE m_csSRWorkingState OF
			
			CELL_WORKING_STATES.e_START:
				fbVirtualCellIntWriter.buffRead := m_sJsonAction; // Inhalt der Datei übergeben
				fbVirtualCellIntWriter.sDestPathName := m_sActionPath; // Pfad der Datei
				fbVirtualCellIntWriter.sDestNetId := m_sAMSNetID;// Net Id des HostPC
				fbVirtualCellIntWriter.tTimeOut := DEFAULT_ADS_TIMEOUT;// Fehlerzeit
				fbVirtualCellIntWriter.bExecute := TRUE;// Positive flanke zum Starten
				IF fbVirtualCellIntWriter.bError THEN//
					m_csCellState := CELL_STATE.e_ERROR;
				END_IF

				m_csSRWorkingState := CELL_WORKING_STATES.e_WORKING;

				
			CELL_WORKING_STATES.e_WORKING:	
				fbVirtualCellIntWriter.bExecute := FALSE; // Nur positive Flanke
				IF NOT(fbVirtualCellIntWriter.bBusy) THEN // Der Funktionsblock aufgehört hat zu arbeiten nächster Schritt ggf. das vorhanden sein der Datei prüfen 
					m_csSRWorkingState := CELL_WORKING_STATES.e_FINISHED;
				END_IF
				
			CELL_WORKING_STATES.e_FINISHED:
				m_iWorkpiece := 0;
				m_sWorkpieceID := 'Empty';
				m_csCellState := CELL_STATE.e_IDEL;
			
		END_CASE
		
	CELL_STATE.e_ERROR:
			;
END_CASE

m_csCellStateLast := m_csCellState;
fbVirtualCellIntWriter();
END_METHOD

END_FUNCTION_BLOCK

// ---- POUs/FB_MHS.TcPOU
FUNCTION_BLOCK FB_MHS
VAR_INPUT
END_VAR
VAR_OUTPUT
END_VAR
VAR
	m_csStateRequest : MHS_STATE;
	m_csStateRequestOld : MHS_STATE;
	m_csState : MHS_STATE;
	m_csStateLastCycle : MHS_STATE;
	m_csStateLastAction : MHS_STATE;
	m_Name : STRING;	
	// Von SystemDemonstratorApp kommend
	m_iWorkpiece : DINT; 
	m_iCell : DINT;
	m_iRequest: DINT;
	// Von SystemDemonstratorApp kommend angenommen
	m_iWorkpieceAccepted : DINT; 
	m_iCellAccepted : DINT;
	m_iRequestAccepted: DINT;
	
	// Von PLC kommend 
	m_iMachineFree : DINT;	
	
	
	//Von MiR kommend
	m_iRequestMachineFree : DINT;
	m_iActionTerminated : DINT;	
	
	
	
	// Zustand der Zelle die Beladen oder Entladen werden soll
	m_eCurrentCellState : CELL_ACTION_STATE;
	m_eNeededCellState : CELL_ACTION_STATE;
	m_bNeededCellStatePending : BOOL;
	
	aMHS : ARRAY [1..20] OF DINT; // Interface API-Array
	
	
	m_iSimulationsTimer : DINT;
END_VAR



StateMachine();

METHOD GetActionFinished : BOOL
VAR_INPUT
END_VAR
IF m_csState = MHS_STATE.e_AKTION_FINISHED THEN
	GetActionFinished := TRUE;
ELSE
	GetActionFinished := FALSE;
END_IF
END_METHOD

METHOD GetCurrentCellForAction : DINT
VAR_INPUT
END_VAR
GetCurrentCellForAction := m_iCellAccepted;
END_METHOD

METHOD GetState : BOOL
VAR_INPUT
END_VAR
END_METHOD

METHOD NeededCellStatePending : BOOL
VAR_INPUT
END_VAR
NeededCellStatePending := m_bNeededCellStatePending;
m_bNeededCellStatePending := FALSE;
END_METHOD

METHOD RequestAction : BOOL
VAR_INPUT
	
	iWorkpiece : DINT; 
	iCell : DINT;
	bRequest : DINT;
END_VAR

m_iWorkpiece :=  iWorkpiece;
m_iCell := iCell;
m_iRequest := bRequest;
END_METHOD

METHOD RequestState : BOOL
VAR_INPUT
END_VAR
END_METHOD

METHOD SendNeededToCell : CELL_ACTION_STATE
VAR_INPUT
END_VAR
SendNeededToCell := m_eNeededCellState;
END_METHOD

METHOD SetClampIsOpen : BOOL
VAR_INPUT
iClampIsOpen : DINT;	

END_VAR
//IF iClampIsOpen > 0 THEN
//	m_iClampIsOpen := 1;
//	m_iClampIsClose := 0;
//ELSE
//	m_iClampIsOpen := 0;
//	m_iClampIsClose := 1;	
//END_IF
END_METHOD

METHOD SetDoorIsOpen : BOOL
VAR_INPUT
	iDoorIsOpen :DINT;
END_VAR
//IF iDoorIsOpen > 0 THEN
//	m_iDoorIsOpen := 1;
//	m_iDoorIsClose := 0;
//ELSE
//	m_iDoorIsOpen := 0;
//	m_iDoorIsClose := 1;	
//END_IF
END_METHOD

METHOD SetMachineFree : BOOL
VAR_INPUT
	iMachineFree:DINT;
END_VAR
m_iMachineFree := iMachineFree;
END_METHOD

METHOD SetStateCurrentMachineForAction : BOOL
VAR_INPUT
	eCurrentCellState :CELL_ACTION_STATE;
END_VAR
m_eCurrentCellState := eCurrentCellState;

SetStateCurrentMachineForAction := TRUE;
END_METHOD


METHOD StateMachine : BOOL
VAR_INPUT
END_VAR

VAR

END_VAR

	// VOM MHS

	{define Simulated}
	//{define MHSConnected}
	
	{IF defined (MHSConnected)}
 	m_iRequestMachineFree   := aMHS[11];
	m_iActionTerminated :=  aMHS[12];
	{END_IF}
	// PLC interne Variablen
	//m_iDoorIsOpen : DINT;	
	//m_iClampIsOpen : DINT;
	//m_iClampIsClose : DINT;	
	//m_iDoorIsClose : DINT;


	
	
CASE m_csState OF

MHS_STATE.e_IDLE: 

	IF m_iWorkpiece > 0 AND m_iCell > 0 AND m_iRequest > 0 THEN
		m_iWorkpieceAccepted := m_iWorkpiece;  
		m_iCellAccepted := m_iCell;
		m_iRequestAccepted:= m_iRequest; 
		m_iWorkpiece := 0;
 		m_iCell := 0;
		m_iRequest := 0;
	
	END_IF

	IF m_iWorkpieceAccepted > 0 AND m_iCellAccepted > 0 AND m_iRequestAccepted = 2 THEN
		aMHS[1] := m_iWorkpiece;
		aMHS[2] := m_iCell;
		aMHS[3] := m_iRequest;
		m_csState := MHS_STATE.e_PGO_POS;	
	END_IF
	IF m_iWorkpieceAccepted > 0 AND m_iCellAccepted > 0 AND m_iRequestAccepted = 1 THEN
		aMHS[1] := m_iWorkpiece;
		aMHS[2] := m_iCell;
		aMHS[3] := m_iRequest;
		m_csState := MHS_STATE.e_GGO_POS;	
	END_IF
	// Löschen dieser Anforderung
	m_iRequestAccepted := 0;



// SUBROUTINE WP in Maschine bringen	  
MHS_STATE.e_PGO_POS:
	
 	IF m_iRequestMachineFree > 0 THEN
		m_eNeededCellState := CELL_ACTION_STATE.e_LoadPos;
		m_bNeededCellStatePending := TRUE;
		m_csState := MHS_STATE.e_PWAIT_DOOR;
	END_IF
	
	{IF defined (Simulated)}
	m_iSimulationsTimer := m_iSimulationsTimer+1;// Simulation	
	IF m_iSimulationsTimer > 1000THEN// Simulation
		m_iSimulationsTimer := 0;// Simulation
		m_iRequestMachineFree := 1;// Simulation
	END_IF// Simulation
	{END_IF}
MHS_STATE.e_PWAIT_DOOR:	
  	IF  m_eCurrentCellState = CELL_ACTION_STATE.e_LoadPos THEN
		m_csState := MHS_STATE.e_PWAIT_CLAMP;
	END_IF
	{IF defined (Simulated)}
	m_iRequestMachineFree := 0;// Simulation
	{END_IF}
MHS_STATE.e_PWAIT_CLAMP:
		m_csState := MHS_STATE.e_PPUT_WP;
	

MHS_STATE.e_PPUT_WP:
		m_csState := MHS_STATE.e_PCLOSE_CLAMP;
 MHS_STATE.e_PCLOSE_CLAMP:
			m_csState := MHS_STATE.e_PLEAFE_MACHINE;	 
MHS_STATE.e_PLEAFE_MACHINE:
 	IF m_iMachineFree > 0 THEN
		m_csState := MHS_STATE.e_AKTION_FINISHED;
	END_IF	
	{IF defined (Simulated)}
	m_iSimulationsTimer := m_iSimulationsTimer + 1;
	IF m_iSimulationsTimer > 1000 THEN// Simulation
		m_iSimulationsTimer := 0;// Simulation
		m_iMachineFree := 1;// Simulation
	END_IF// Simulation
	{END_IF}
// SUBROUTINE WP aus Maschine holen	  
MHS_STATE.e_GGO_POS:
 	IF m_iRequestMachineFree > 0 THEN
		m_eNeededCellState := CELL_ACTION_STATE.e_UnLoadPos;
		m_bNeededCellStatePending := TRUE;
		m_csState := MHS_STATE.e_GWAIT_DOOR;
	END_IF
	{IF defined (Simulated)}
	m_iSimulationsTimer := m_iSimulationsTimer+1;// Simulation	
	
	IF m_iSimulationsTimer > 1000THEN// Simulation
		m_iSimulationsTimer := 0;// Simulation
		m_iRequestMachineFree := 1;// Simulation
	END_IF// Simulation
	{END_IF}
	
MHS_STATE.e_GWAIT_DOOR:
  	IF  m_eCurrentCellState = CELL_ACTION_STATE.e_UnLoadPos THEN
		m_csState := MHS_STATE.e_GWAIT_CLAMP;
	END_IF
	{IF defined (Simulated)}
		m_iRequestMachineFree := 0;// Simulation
	{END_IF}
MHS_STATE.e_GWAIT_CLAMP:
	//IF m_iClampIsOpen > 0 THEN
		m_csState := MHS_STATE.e_GGET_WP;
	//END_IF
MHS_STATE.e_GGET_WP:
	//IF 	m_iClampCloseRequest > 0 THEN
		m_csState := MHS_STATE.e_GCLOSE_CLAMP;
	//END_IF
 MHS_STATE.e_GCLOSE_CLAMP:
 	//IF m_iClampIsClose > 0 THEN
			m_csState := MHS_STATE.e_GLEAFE_MACHINE;	 
 	//END_IF
MHS_STATE.e_GLEAFE_MACHINE:
 	IF m_iMachineFree > 0 THEN
		m_csState := MHS_STATE.e_AKTION_FINISHED;
	END_IF		
	{IF defined (Simulated)}
	m_iSimulationsTimer := m_iSimulationsTimer + 1;
	IF m_iSimulationsTimer > 1000 THEN// Simulation
		m_iSimulationsTimer := 0;// Simulation
		m_iMachineFree := 1;// Simulation
	END_IF// Simulation
	{END_IF}
MHS_STATE.e_AKTION_FINISHED:
	m_csState := MHS_STATE.e_IDLE;
	m_iMachineFree := 0;
	
MHS_STATE.e_ERROR:
	
ELSE
	m_csState := MHS_STATE.e_ERROR;
 
END_CASE
{IF defined (MHSConnected)}
m_iMachineFree := aMHS[4];
{END_IF}
END_METHOD

END_FUNCTION_BLOCK

// ---- POUs/FB_Clamp.TcPOU
FUNCTION_BLOCK FB_Clamp
VAR_INPUT
	
END_VAR
VAR_OUTPUT
END_VAR
VAR
m_csState : CLAMP_STATE;	
m_csStateRequested : CLAMP_STATE;

//Eingänge
m_bIsOpen : BOOL;
m_bIsClosed : BOOL;
m_bIsClosedFull : BOOL;

//Ausgänge
m_bOpen :BOOL;
m_bClose :BOOL;

END_VAR


StateMachine();

METHOD IsClosed : BOOL
VAR_INPUT
END_VAR
IF m_csState = CLAMP_STATE.e_CLOSED THEN
	IsClosed := TRUE;
END_IF
END_METHOD

METHOD IsClosedFull : BOOL
VAR_INPUT
END_VAR
IF m_csState = CLAMP_STATE.e_CLOSED_FULL THEN
	IsClosedFull := TRUE;
END_IF
END_METHOD

METHOD IsError : BOOL
VAR_INPUT
END_VAR
IF m_csState = CLAMP_STATE.e_ERROR THEN
	IsError := TRUE;
END_IF
END_METHOD

METHOD IsOpen : BOOL
VAR_INPUT
END_VAR
IF m_csState = CLAMP_STATE.e_OPEN THEN
	IsOpen := TRUE;
END_IF
END_METHOD

METHOD SetCloseClampEmpty : BOOL
VAR_INPUT
END_VAR
m_csStateRequested := CLAMP_STATE.e_CLOSED;
m_bClose := TRUE;
SetCloseClampEmpty:=TRUE;
END_METHOD

METHOD SetCloseClampFull : BOOL
VAR_INPUT
END_VAR
m_csStateRequested := CLAMP_STATE.e_CLOSED_FULL;
m_bClose := TRUE;
SetCloseClampFull := TRUE;
END_METHOD

METHOD SetOpenClamp : BOOL
VAR_INPUT
END_VAR
m_bOpen := TRUE;
END_METHOD

METHOD StateMachine : BOOL
VAR_INPUT
END_VAR

//m_bIsOpen : BOOL;
//m_bIsClosed : BOOL;
//m_bIsClosedFull : BOOL;

CASE m_csState  OF
	
	CLAMP_STATE.e_OPEN:	
		

		IF m_bIsClosed THEN
			m_csState := CLAMP_STATE.e_CLOSED;		
		END_IF
		
		IF m_bIsClosedFull THEN
			m_csState := CLAMP_STATE.e_CLOSED_FULL;		
		END_IF
		
 	CLAMP_STATE.e_CLOSED_FULL:
	// Fehler wenn falscher Zustand
 		IF m_csStateRequested = CLAMP_STATE.e_CLOSED THEN
  			m_csState := CLAMP_STATE.e_ERROR;
		END_IF
		
		
		IF m_bIsOpen THEN
			m_csState := CLAMP_STATE.e_OPEN;		
		END_IF
	
	CLAMP_STATE.e_CLOSED:
			// Fehler wenn falscher Zustand in diesem Fall: Werkstück erwartet aber nicht im Halter
 		IF m_csStateRequested = CLAMP_STATE.e_CLOSED_FULL THEN
  			m_csState := CLAMP_STATE.e_ERROR;
		END_IF
	
	
		IF m_bIsOpen THEN
			m_csState := CLAMP_STATE.e_OPEN;		
		END_IF
		
CLAMP_STATE.e_ERROR:
		
END_CASE
END_METHOD

END_FUNCTION_BLOCK

// ---- POUs/FB_InterfaceIO.TcPOU
FUNCTION_BLOCK FB_InterfaceIO IMPLEMENTS ITF_Cell
VAR_INPUT

END_VAR
VAR_OUTPUT
END_VAR

VAR
	// Ausgang :engine          AT %IX0.0:        BOOL; 
//Eingänge
//A5Q_Bestuckung AT %QX27.4 : BOOL;
//A5Q_Startfreigabe AT %QX27.5 : BOOL;
//A5Q_Entnahme AT %QX27.6 : BOOL;
//A5Q_Standby AT %QX27.7 : BOOL;
//A5Q_NOT_Aus_Befehl AT %QX28.0 : BOOL;

//INPUTS  A5 Station Variabel : 5V Von Arduino

//A5I_Bestuckbereit_o1 AT %IX43.2 : BOOL;  
//A5I_Arbeitet_o2 AT %IX43.3 : BOOL;
//A5I_Fertig_o3 AT %IX43.4 : BOOL;
//A5I_Storung_o5 AT %IX43.5 : BOOL;
//A5I_NOT_Halt_o6 AT %IX43.6 : BOOL;
//A5I_Pro_Standby_o7 AT %IX43.7 : BOOL;
//A5I_Pro_Standby_o8 AT %IX44.0 : BOOL;
 
m_bEmergencyOff AT %IX43.6 : BOOL;
m_bEmergencyStop AT %IX43.5 : BOOL;
m_bFinished AT %IX43.4 : BOOL;
m_bRunning AT %IX43.3 : BOOL;
m_bLoadPos  AT %IX43.2 : BOOL; 
m_bUnloadPos  AT %IX43.2 : BOOL; 
m_bStandby AT %IX44.0 : BOOL;
m_bStartable AT %IX43.7 : BOOL;
// Ausgang :engine          AT %QX0.0:        BOOL; 
// Ausgänge
m_bToEmergencyOff AT %QX28.0 : BOOL;
m_bToEmergencyStop AT %QX28.0 : BOOL;
m_bMoveToLoadPos AT %QX27.4 : BOOL;
m_bMoveToUnloadPos AT %QX27.4 : BOOL;
m_bToStandby AT %QX27.7 : BOOL;
m_bStart AT %QX27.5 : BOOL;

END_VAR

// Logik des Interfaces in diesem Fall zurücksetzen der Ausgänge nach erreichen des Ziels 
// Aus Zustandsmaschine Löschen ggf. ??
IF m_bEmergencyOff THEN
m_bToEmergencyOff := FALSE;
END_IF

IF m_bEmergencyStop THEN
m_bToEmergencyStop := FALSE;
END_IF

IF m_bLoadPos THEN
	m_bMoveToLoadPos := FALSE;
END_IF

IF m_bUnloadPos THEN
	m_bMoveToUnloadPos := FALSE;
END_IF

IF m_bStandby THEN
	m_bToStandby := FALSE;
END_IF

IF m_bRunning THEN
	m_bStart := FALSE;
END_IF

METHOD GetEmergencyOff : BOOL
VAR_INPUT
END_VAR
GetEmergencyOff := m_bEmergencyOff;
END_METHOD

METHOD GetEmergencyStop : BOOL
VAR_INPUT
END_VAR
GetEmergencyStop := m_bEmergencyStop;
END_METHOD

METHOD GetFinished : BOOL
VAR_INPUT
END_VAR
GetFinished := m_bFinished;
END_METHOD

METHOD GetIsRunning : BOOL
VAR_INPUT
END_VAR
GetIsRunning := m_bRunning;
END_METHOD

METHOD GetLoadPos : BOOL
VAR_INPUT
END_VAR
GetLoadPos := m_bLoadPos;
END_METHOD

METHOD GetStandby : BOOL
VAR_INPUT
END_VAR
GetStandby := m_bStandby;
END_METHOD

METHOD GetStartable : BOOL
VAR_INPUT
END_VAR
GetStartable := m_bStartable;
END_METHOD

METHOD GetUnloadPos : BOOL
VAR_INPUT
END_VAR
GetUnloadPos := m_bUnloadPos;
END_METHOD

METHOD SetEmergencyOff : BOOL
VAR_INPUT
	b :BOOL;
END_VAR

m_bToEmergencyOff := b;
SetEmergencyOff:=b;
END_METHOD

METHOD SetEmergencyStop : BOOL
VAR_INPUT
	b :BOOL;
END_VAR
m_bToEmergencyStop :=b;

SetEmergencyStop := b;
END_METHOD

METHOD SetMoveToLoad : BOOL
VAR_INPUT
	b :BOOL;
END_VAR
m_bMoveToLoadPos := b;

SetMoveToLoad := b;
END_METHOD

METHOD SetMoveToUnload : BOOL
VAR_INPUT
	b :BOOL;
END_VAR
m_bMoveToUnloadPos := b;

SetMoveToUnload := b;
END_METHOD

METHOD SetStandby : BOOL
VAR_INPUT
	b :BOOL;
END_VAR
m_bToStandby := b;

SetStandby := b;
END_METHOD

METHOD SetStart : BOOL
VAR_INPUT
	b :BOOL;
END_VAR
m_bStart := b;

SetStart := b;
END_METHOD

END_FUNCTION_BLOCK

// ---- POUs/POU.TcPOU
FUNCTION_BLOCK POU
VAR_INPUT
END_VAR
VAR_OUTPUT
END_VAR
VAR
END_VAR

END_FUNCTION_BLOCK
